Fanuc KAREL source: kt00375.KL

-- PROVISIONAL review KL for V1013-1; original PC SHA256 62f149c6247f5cdaab269f5d6928ac4686ac7bf23f8034bb1b7cf672f42e6985
-- Incomplete behavior may be omitted. Consult companion uncertainty JSON. Do not deploy.
PROGRAM KT00375
%NOLOCKGROUP
VAR
  I2 : INTEGER
  OUT : BOOLEAN
-- UNRESOLVED_DECL Y1 type=002018
BEGIN
  -- UNRESOLVED_PC offsets 5-19; opcodes 2E,22,9D,33,B2
  -- UNRESOLVED_PC offsets 24-35; opcodes 2E,23
  -- UNRESOLVED_PC offsets 40-62; opcodes 22,9D,33,B1,21,5A,23
  -- UNRESOLVED_PC offsets 67-71; opcodes 7F
END KT00375
